PROGRAM MAIN
VAR
	testPid_ : BOOL := FALSE;
	testController_ : PidControllerTest;
END_VAR


IF testPid_ THEN
	testController_.cyclic();
ELSE
	testController_.reset();
END_IF

END_PROGRAM

(* stored: Version 1.1.0.1, ProductVersion 3.1.4026.6
   POU MAIN: Id {08b7b4be-dd7c-4968-925b-b68dd8a83ed1}, SpecialFunc None *)
